(* LS Electric XG5000 project: AIR_PRESSURE_CONTROL_USING_PLC_04_06 *)
(* PLC LSPLC *)
(* module base 0 slot 0: Input/Output Module:XEC-DR32H (DC 24V input 16 points, relay output 16 points) *)
(* module base 0 slot 1: Analog IO Module:XBF-AH04A (A/D Voltage/Current 2 Ch, D/A Voltage/Current 2 Ch) *)
VAR_GLOBAL
    LOAD AT %QX0.0.1 : BOOL;
    OUT_DATA : WORD;
    _01_AD01_DATA_ARY AT %UW0.1.4 : ARRAY[0..1] OF WORD; (* Analog IO Module: Input each CH Data *)
    _01_AD0_DATA AT %UW0.1.4 : WORD; (* Analog IO Module: AD0 Digital Output Data *)
    _01_DA0_ACT AT %UX0.1.18 : BOOL; (* Analog IO Module: DA0 Activation Status *)
    _01_DA_OUTEN_ARY AT %UX0.1.96 : ARRAY[0..1] OF BOOL; (* Analog IO Module: Output each CH Status Setting *)
END_VAR

PROGRAM NewProgram (* task: Scan Program *)
VAR_EXTERNAL
    LOAD : BOOL; (* AT %QX0.0.1 *)
    OUT_DATA : WORD;
    _01_AD01_DATA_ARY : ARRAY[0..1] OF WORD; (* AT %UW0.1.4 *) (* Analog IO Module: Input each CH Data *)
    _01_AD0_DATA : WORD; (* AT %UW0.1.4 *) (* Analog IO Module: AD0 Digital Output Data *)
    _01_DA0_ACT : BOOL; (* AT %UX0.1.18 *) (* Analog IO Module: DA0 Activation Status *)
    _01_DA_OUTEN_ARY : ARRAY[0..1] OF BOOL; (* AT %UX0.1.96 *) (* Analog IO Module: Output each CH Status Setting *)
END_VAR

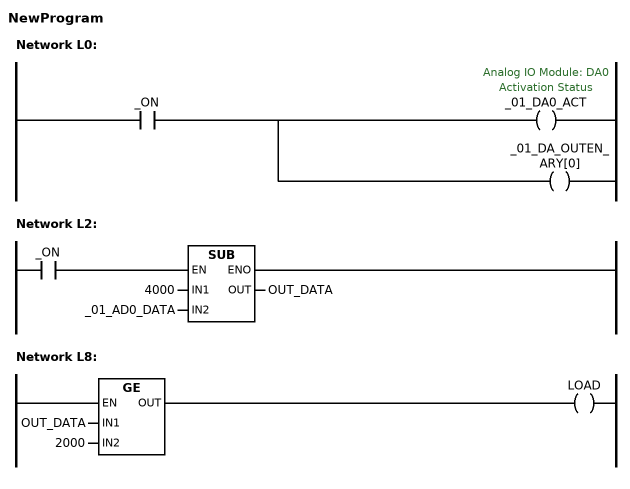
(* Rung L0 *)
_01_DA0_ACT := _ON;
_01_DA_OUTEN_ARY[0] := _ON;
(* Rung L2 *)
IF _ON THEN OUT_DATA := 4000 - _01_AD0_DATA; END_IF;
(* Rung L8 *)
LOAD := OUT_DATA >= 2000;
END_PROGRAM